FUNCTION CalculateAverage : REAL
VAR_INPUT
	 arrMarks : ARRAY[1..20] OF REAL;
END_VAR
VAR
	 i : INT;
    sum : REAL := 0;
END_VAR


FOR i := 1 TO 10 DO
    sum := sum + arrMarks[i];
END_FOR

CalculateAverage := sum / 20;

END_FUNCTION

(* stored: Version 1.1.0.1, ProductVersion 3.1.4024.16
   POU CalculateAverage: Id {7dc42628-96fc-4b72-97b9-0f9d0b5a9bca}, SpecialFunc None *)
